(* IEC 61131-3 sources: tuk_project/src/control_systems/modelling/split_section_models, 2 files *)

(* ---- production.st ---- *)
PROGRAM program0

(*=====================================================================*)
(*DECLARATION*)
(*=====================================================================*)

VAR

(*INPUTS*)
S_AL1_P_B1 AT %IX100.0 : BOOL;
S_AL1_P_B2 AT %IX100.1 : BOOL;
S_AL1_MCB AT %IX100.2 : BOOL;
MCB_BUSY AT %IX100.3 : BOOL;
S_AL1_MCBR AT %IX100.4 : BOOL;
MCBR_BUSY AT %IX100.5 : BOOL;
S_AL1_MCB2 AT %IX100.6 : BOOL;
S_AL1_MCBR2 AT %IX100.7 : BOOL;
E_AL1_B1 AT %QX100.0 : BOOL;
PUWS_AL1_B1_PLUS AT %QX100.1 : BOOL;
PUWS_AL1_B1_RIGHT AT %QX100.2 : BOOL;
PAS_AL1_PLUS AT %QX100.3 : BOOL;
PAS_AL1_TURN AT %QX100.4 : BOOL;

END_VAR

VAR

(*PLACES*)

PPAL1 : BOOL := 1;
PP0 : BOOL := 1;
PP1 : BOOL := 0;
PP2 : BOOL := 0;
PP3 : BOOL := 0;
PP4 : BOOL := 0;
MCB : BOOL := 1;
PP5 : BOOL := 0;
PP7 : BOOL := 0;
PPL3 : BOOL := 0;
PPL4 : BOOL := 0;
MCBR : BOOL := 1;
PPL5 : BOOL := 0;
PPL7 : BOOL := 0;
STABLE : BOOL := 0;

END_VAR

VAR

(*INTERNAL VARIABLES*)

MCB_CONTROL : BOOL;

END_VAR

(*=====================================================================*)
(*TRANSITIONS*)
(*=====================================================================*)

STABLE:=0;
WHILE STABLE=0 DO
   STABLE:=1;
   (*TP0*)
   IF (PP0) AND ( (NOT MCB_CONTROL) ) AND (NOT PP1) THEN
       PP0:=0;
       PP1:=1;
       STABLE:=0;
   END_IF;
   (*TP1*)
   IF (PP1) AND ( (S_AL1_P_B1) ) AND (NOT PP2) THEN
       PP1:=0;
       PP2:=1;
       STABLE:=0;
   END_IF;
   (*TP2*)
   IF (PP2) AND ( (S_AL1_P_B2 AND NOT MCB_CONTROL) ) AND (NOT PP3) THEN
       PP2:=0;
       PP3:=1;
       STABLE:=0;
   END_IF;
   (*TP3*)
   IF (PP3) AND ( (S_AL1_MCB) ) AND (NOT PP4 AND NOT PP1) THEN
       PP3:=0;
       PP4:=1;
       PP1:=1;
       STABLE:=0;
   END_IF;
   (*TP4*)
   IF (PP4 AND MCB) AND ( (MCB_BUSY) ) AND (NOT PP5) THEN
       PP4:=0;
       MCB:=0;
       PP5:=1;
       STABLE:=0;
   END_IF;
   (*TP6*)
   IF (PP5) AND ( (S_AL1_MCB2) ) AND (NOT PP7 AND NOT MCB) THEN
       PP5:=0;
       PP7:=1;
       MCB:=1;
       STABLE:=0;
   END_IF;
   (*TPL2*)
   IF (PP2) AND ( (S_AL1_P_B2 AND MCB_CONTROL) ) AND (NOT PPL3 AND NOT PP1) THEN
       PP2:=0;
       PPL3:=1;
       PP1:=1;
       STABLE:=0;
   END_IF;
   (*TPL3*)
   IF (PPL3) AND ( (S_AL1_MCBR) ) AND (NOT PPL4) THEN
       PPL3:=0;
       PPL4:=1;
       STABLE:=0;
   END_IF;
   (*TPL4*)
   IF (PPL4 AND MCBR) AND ( (MCBR_BUSY) ) AND (NOT PPL5) THEN
       PPL4:=0;
       MCBR:=0;
       PPL5:=1;
       STABLE:=0;
   END_IF;
   (*TPL6*)
   IF (PPL5) AND ( (S_AL1_MCBR2) ) AND (NOT PPL7 AND NOT MCBR) THEN
       PPL5:=0;
       PPL7:=1;
       MCBR:=1;
       STABLE:=0;
   END_IF;
END_WHILE;

(*=====================================================================*)
(*OUTPUTS*)
(*=====================================================================*)

(*E_AL1_B1*)
IF PP0 OR PP1 THEN
   E_AL1_B1:=1;
END_IF;
(*MCB_CONTROL*)
IF PP3 THEN
   MCB_CONTROL:=1;
END_IF;
(*PAS_AL1_PLUS*)
IF PPL3 OR PPL4 THEN
   PAS_AL1_PLUS:=1;
END_IF;
(*PAS_AL1_TURN*)
IF PPL3 OR PPL4 THEN
   PAS_AL1_TURN:=1;
END_IF;
(*PUWS_AL1_B1_PLUS*)
IF PPAL1 OR PP2 THEN
   PUWS_AL1_B1_PLUS:=1;
END_IF;
(*E_AL1_B1*)
IF PP2 OR PP3 OR PPL3 THEN
   E_AL1_B1:=0;
END_IF;
(*MCB_CONTROL*)
IF PP0 OR PPL3 THEN
   MCB_CONTROL:=0;
END_IF;
(*PAS_AL1_PLUS*)
IF PP0 OR PP3 OR PP4 THEN
   PAS_AL1_PLUS:=0;
END_IF;
(*PAS_AL1_TURN*)
IF PP0 OR PP3 OR PP4 THEN
   PAS_AL1_TURN:=0;
END_IF;
(*PUWS_AL1_B1_RIGHT*)
IF PPAL1 OR PP2 THEN
   PUWS_AL1_B1_RIGHT:=0;
END_IF;

END_PROGRAM

CONFIGURATION config0

    RESOURCE res0 ON PLC
        TASK task0(INTERVAL := T#20ms, PRIORITY := 0);
        PROGRAM instance0 WITH task0 : program0;
    END_RESOURCE

END_CONFIGURATION

(* ---- storage_model.st ---- *)
PROGRAM program0

(*=====================================================================*)
(*DECLARATION*)
(*=====================================================================*)

VAR

(*INPUTS*)
AL1_G_S1 AT %IX100.0 : BOOL;
AL1_G_SC_LL AT %IX100.1 : BOOL;
AL1_G_SC_MZ AT %IX100.2 : BOOL;
AL1_G_ML AT %IX100.3 : BOOL;
AL1_G_SC_MX AT %IX100.4 : BOOL;
AL1_G_SC_RL AT %IX100.5 : BOOL;
RC_AL1_G7 AT %QX100.0 : BOOL;
AL1_G_SC_LT AT %QX100.1 : BOOL;
AL1_G_SC_LIFT AT %QX100.2 : BOOL;
AL1_G_SC_RT AT %QX100.3 : BOOL;
AL1_G_SC_TG AT %QW100 : INT;

END_VAR

VAR

(*PLACES*)

PG0 : BOOL := 0;
PG : BOOL := 1;
PG1 : BOOL := 0;
PG2 : BOOL := 0;
PG3 : BOOL := 0;
PG4 : BOOL := 0;
PG5 : BOOL := 0;
PG6 : BOOL := 0;
PG7 : BOOL := 0;
PG8 : BOOL := 0;
PG9 : BOOL := 0;
PG10 : BOOL := 0;
PG11 : BOOL := 0;
PG12 : BOOL := 0;
PG13 : BOOL := 0;
PG14 : BOOL := 0;
PG15 : BOOL := 0;
PG16 : BOOL := 0;
PG17 : BOOL := 0;
PG18 : BOOL := 0;
PG19 : BOOL := 0;
PG20 : BOOL := 0;
PG21 : BOOL := 0;
PG22 : BOOL := 0;
PG23 : BOOL := 0;
PG24 : BOOL := 0;
PG25 : BOOL := 0;
PG26 : BOOL := 0;
STABLE : BOOL := 0;

END_VAR

VAR

(*INTERNAL VARIABLES*)

TG_POS : INT;

END_VAR

TG_POS:=10;

(*=====================================================================*)
(*TRANSITIONS*)
(*=====================================================================*)

STABLE:=0;
WHILE STABLE=0 DO
   STABLE:=1;
   (*TG1*)
   IF (PG AND PG0) AND ( (NOT AL1_G_S1) ) AND (NOT PG1) THEN
       PG:=0;
       PG0:=0;
       PG1:=1;
       STABLE:=0;
   END_IF;
   (*TG2*)
   IF (PG1) AND ( (AL1_G_SC_LL) ) AND (NOT PG2) THEN
       PG1:=0;
       PG2:=1;
       STABLE:=0;
   END_IF;
   (*TG3*)
   IF (PG2) AND ( (AL1_G_SC_MZ) ) AND (NOT PG3) THEN
       PG2:=0;
       PG3:=1;
       STABLE:=0;
   END_IF;
   (*TG4*)
   IF (PG3) AND ( (NOT AL1_G_SC_MZ) ) AND (NOT PG4) THEN
       PG3:=0;
       PG4:=1;
       STABLE:=0;
   END_IF;
   (*TG5*)
   IF (PG4) AND ( (AL1_G_ML) ) AND (NOT PG5) THEN
       PG4:=0;
       PG5:=1;
       STABLE:=0;
   END_IF;
   (*TG6*)
   IF (PG5) AND ( (AL1_G_SC_MZ) ) AND (NOT PG6) THEN
       PG5:=0;
       PG6:=1;
       STABLE:=0;
   END_IF;
   (*TG7*)
   IF (PG6) AND ( (NOT AL1_G_SC_MZ) ) AND (NOT PG7) THEN
       PG6:=0;
       PG7:=1;
       STABLE:=0;
   END_IF;
   (*TG8*)
   IF (PG7) AND ( (TRUE) ) AND (NOT PG8 AND NOT PG11) THEN
       PG7:=0;
       PG8:=1;
       PG11:=1;
       STABLE:=0;
   END_IF;
   (*TG9*)
   IF (PG8) AND ( (AL1_G_SC_MX) ) AND (NOT PG9) THEN
       PG8:=0;
       PG9:=1;
       STABLE:=0;
   END_IF;
   (*TG10*)
   IF (PG9) AND ( (NOT AL1_G_SC_MX) ) AND (NOT PG10) THEN
       PG9:=0;
       PG10:=1;
       STABLE:=0;
   END_IF;
   (*TG12*)
   IF (PG11) AND ( (AL1_G_SC_MZ) ) AND (NOT PG12) THEN
       PG11:=0;
       PG12:=1;
       STABLE:=0;
   END_IF;
   (*TG13*)
   IF (PG12) AND ( (NOT AL1_G_SC_MZ) ) AND (NOT PG13) THEN
       PG12:=0;
       PG13:=1;
       STABLE:=0;
   END_IF;
   (*TG14*)
   IF (PG10 AND PG13) AND ( (TRUE) ) AND (NOT PG14) THEN
       PG10:=0;
       PG13:=0;
       PG14:=1;
       STABLE:=0;
   END_IF;
   (*TG15*)
   IF (PG14) AND ( (AL1_G_SC_MZ) ) AND (NOT PG15) THEN
       PG14:=0;
       PG15:=1;
       STABLE:=0;
   END_IF;
   (*TG16*)
   IF (PG15) AND ( (NOT AL1_G_SC_MZ) ) AND (NOT PG16) THEN
       PG15:=0;
       PG16:=1;
       STABLE:=0;
   END_IF;
   (*TG17*)
   IF (PG16) AND ( (AL1_G_SC_RL) ) AND (NOT PG17) THEN
       PG16:=0;
       PG17:=1;
       STABLE:=0;
   END_IF;
   (*TG18*)
   IF (PG17) AND ( (AL1_G_SC_MZ) ) AND (NOT PG18) THEN
       PG17:=0;
       PG18:=1;
       STABLE:=0;
   END_IF;
   (*TG19*)
   IF (PG18) AND ( (NOT AL1_G_SC_MZ) ) AND (NOT PG19) THEN
       PG18:=0;
       PG19:=1;
       STABLE:=0;
   END_IF;
   (*TG20*)
   IF (PG19) AND ( (AL1_G_ML) ) AND (NOT PG20) THEN
       PG19:=0;
       PG20:=1;
       STABLE:=0;
   END_IF;
   (*TG21*)
   IF (PG20) AND ( (TRUE) ) AND (NOT PG21 AND NOT PG24) THEN
       PG20:=0;
       PG21:=1;
       PG24:=1;
       STABLE:=0;
   END_IF;
   (*TG22*)
   IF (PG21) AND ( (AL1_G_SC_MX) ) AND (NOT PG22) THEN
       PG21:=0;
       PG22:=1;
       STABLE:=0;
   END_IF;
   (*TG23*)
   IF (PG22) AND ( (NOT AL1_G_SC_MX) ) AND (NOT PG23) THEN
       PG22:=0;
       PG23:=1;
       STABLE:=0;
   END_IF;
   (*TG25*)
   IF (PG24) AND ( (AL1_G_SC_MZ) ) AND (NOT PG25) THEN
       PG24:=0;
       PG25:=1;
       STABLE:=0;
   END_IF;
   (*TG26*)
   IF (PG25) AND ( (NOT AL1_G_SC_MZ) ) AND (NOT PG26) THEN
       PG25:=0;
       PG26:=1;
       STABLE:=0;
   END_IF;
   (*TG27*)
   IF (PG23 AND PG26) AND ( (TRUE) ) AND (NOT PG) THEN
       PG23:=0;
       PG26:=0;
       PG:=1;
       STABLE:=0;
   END_IF;
END_WHILE;

(*=====================================================================*)
(*OUTPUTS*)
(*=====================================================================*)

(*AL1_G_SC_LIFT*)
IF PG2 OR PG3 OR PG4 OR PG14 OR PG15 OR PG16 THEN
   AL1_G_SC_LIFT:=1;
END_IF;
(*AL1_G_SC_LT*)
IF PG1 OR PG2 OR PG3 THEN
   AL1_G_SC_LT:=1;
END_IF;
(*AL1_G_SC_RT*)
IF PG16 OR PG17 OR PG18 THEN
   AL1_G_SC_RT:=1;
END_IF;
(*RC_AL1_G7*)
IF PG THEN
   RC_AL1_G7:=1;
END_IF;
(*AL1_G_SC_LIFT*)
IF PG OR PG1 OR PG5 OR PG6 OR PG7 OR PG8 OR PG9 OR PG10 OR PG11 OR PG12 OR PG13 OR PG17 OR PG18 OR PG19 OR PG20 OR PG21 OR PG22 OR PG23 OR PG24 OR PG25 OR PG26 THEN
   AL1_G_SC_LIFT:=0;
END_IF;
(*AL1_G_SC_LT*)
IF PG OR PG4 OR PG5 OR PG6 OR PG7 OR PG8 OR PG9 OR PG10 OR PG11 OR PG12 OR PG13 OR PG14 OR PG15 OR PG16 OR PG17 OR PG18 OR PG19 OR PG20 OR PG21 OR PG22 OR PG23 OR PG24 OR PG25 OR PG26 THEN
   AL1_G_SC_LT:=0;
END_IF;
(*AL1_G_SC_RT*)
IF PG OR PG1 OR PG2 OR PG3 OR PG4 OR PG5 OR PG6 OR PG7 OR PG8 OR PG9 OR PG10 OR PG11 OR PG12 OR PG13 OR PG14 OR PG15 OR PG19 OR PG20 OR PG21 OR PG22 OR PG23 OR PG24 OR PG25 OR PG26 THEN
   AL1_G_SC_RT:=0;
END_IF;
(*RC_AL1_G7*)
IF PG1 OR PG2 OR PG3 OR PG4 OR PG5 OR PG6 OR PG7 OR PG8 OR PG9 OR PG10 OR PG11 OR PG12 OR PG13 OR PG14 OR PG15 OR PG16 OR PG17 OR PG18 OR PG19 OR PG20 OR PG21 OR PG22 OR PG23 OR PG24 OR PG25 OR PG26 THEN
   RC_AL1_G7:=0;
END_IF;
(*AL1_G_SC_TG*)
IF PG THEN
   AL1_G_SC_TG:=55;
END_IF;
(*AL1_G_SC_TG*)
IF PG1 THEN
   AL1_G_SC_TG:=55;
END_IF;
(*AL1_G_SC_TG*)
IF PG2 THEN
   AL1_G_SC_TG:=55;
END_IF;
(*AL1_G_SC_TG*)
IF PG3 THEN
   AL1_G_SC_TG:=55;
END_IF;
(*AL1_G_SC_TG*)
IF PG4 THEN
   AL1_G_SC_TG:=55;
END_IF;
(*AL1_G_SC_TG*)
IF PG5 THEN
   AL1_G_SC_TG:=55;
END_IF;
(*AL1_G_SC_TG*)
IF PG6 THEN
   AL1_G_SC_TG:=55;
END_IF;
(*AL1_G_SC_TG*)
IF PG7 THEN
   AL1_G_SC_TG:=TG_POS;
END_IF;
(*AL1_G_SC_TG*)
IF PG8 THEN
   AL1_G_SC_TG:=TG_POS;
END_IF;
(*AL1_G_SC_TG*)
IF PG9 THEN
   AL1_G_SC_TG:=TG_POS;
END_IF;
(*AL1_G_SC_TG*)
IF PG10 THEN
   AL1_G_SC_TG:=TG_POS;
END_IF;
(*AL1_G_SC_TG*)
IF PG11 THEN
   AL1_G_SC_TG:=TG_POS;
END_IF;
(*AL1_G_SC_TG*)
IF PG12 THEN
   AL1_G_SC_TG:=TG_POS;
END_IF;
(*AL1_G_SC_TG*)
IF PG13 THEN
   AL1_G_SC_TG:=TG_POS;
END_IF;
(*AL1_G_SC_TG*)
IF PG14 THEN
   AL1_G_SC_TG:=TG_POS;
END_IF;
(*AL1_G_SC_TG*)
IF PG15 THEN
   AL1_G_SC_TG:=TG_POS;
END_IF;
(*AL1_G_SC_TG*)
IF PG16 THEN
   AL1_G_SC_TG:=TG_POS;
END_IF;
(*AL1_G_SC_TG*)
IF PG17 THEN
   AL1_G_SC_TG:=TG_POS;
END_IF;
(*AL1_G_SC_TG*)
IF PG18 THEN
   AL1_G_SC_TG:=TG_POS;
END_IF;
(*AL1_G_SC_TG*)
IF PG19 THEN
   AL1_G_SC_TG:=TG_POS;
END_IF;
(*AL1_G_SC_TG*)
IF PG20 THEN
   AL1_G_SC_TG:=55;
END_IF;
(*AL1_G_SC_TG*)
IF PG21 THEN
   AL1_G_SC_TG:=55;
END_IF;
(*AL1_G_SC_TG*)
IF PG22 THEN
   AL1_G_SC_TG:=55;
END_IF;
(*AL1_G_SC_TG*)
IF PG23 THEN
   AL1_G_SC_TG:=55;
END_IF;
(*AL1_G_SC_TG*)
IF PG24 THEN
   AL1_G_SC_TG:=55;
END_IF;
(*AL1_G_SC_TG*)
IF PG25 THEN
   AL1_G_SC_TG:=55;
END_IF;
(*AL1_G_SC_TG*)
IF PG26 THEN
   AL1_G_SC_TG:=55;
END_IF;

END_PROGRAM

CONFIGURATION config0

    RESOURCE res0 ON PLC
        TASK task0(INTERVAL := T#20ms, PRIORITY := 0);
        PROGRAM instance0 WITH task0 : program0;
    END_RESOURCE

END_CONFIGURATION
